// TIA Portal V17 export
// export: Created 2025-03-05T08:03:02.5022413Z, ExportSetting WithDefaults, DisplayName Totally Integrated Automation Portal, DisplayVersion V17 Update 8, DisplayName TIA Portal Openness, DisplayVersion V17 Update 8, DisplayName TIA Portal Version Control Interface, DisplayVersion V17, DisplayName SINAMICS Startdrive Advanced, DisplayVersion V17 SP2, DisplayName SINAMICS Startdrive G110M, G120, G120C, G120D, G120P, G115D, DisplayVersion V17 SP2, DisplayName SINAMICS Startdrive G130, G150, S120, S150, SINAMICS MV, S210, DisplayVersion V17 SP2, DisplayName STEP 7 Professional, DisplayVersion V17 Update 8, DisplayName SINUMERIK ONE STEP 7 Toolbox, DisplayVersion V17 Update 12, DisplayName SINUMERIK 840D sl STEP 7 Toolbox, DisplayVersion V17 Update 12, DisplayName STEP 7 Safety, DisplayVersion V17 Update 6, DisplayName WinCC Advanced, DisplayVersion V17 Update 8
FUNCTION "FC21012_POWDER_FEEDER_HEATER_JKL" : Void   // FC21012, LAD
TITLE = FC21012 POWDER FEEDER HEATER JKL
{ S7_Optimized_Access := 'TRUE' }
VERSION : 0.1
// stored: AutoNumber false, IsIECCheckEnabled false, SetENOAutomatically false, UDAEnableTagReadback false
BEGIN

REGION Network 1: /////_UNIT_01_/////
END_REGION

REGION Network 2: CALL FB21012 POWDER FEEDER 1 HEATER JKL UNIT 01
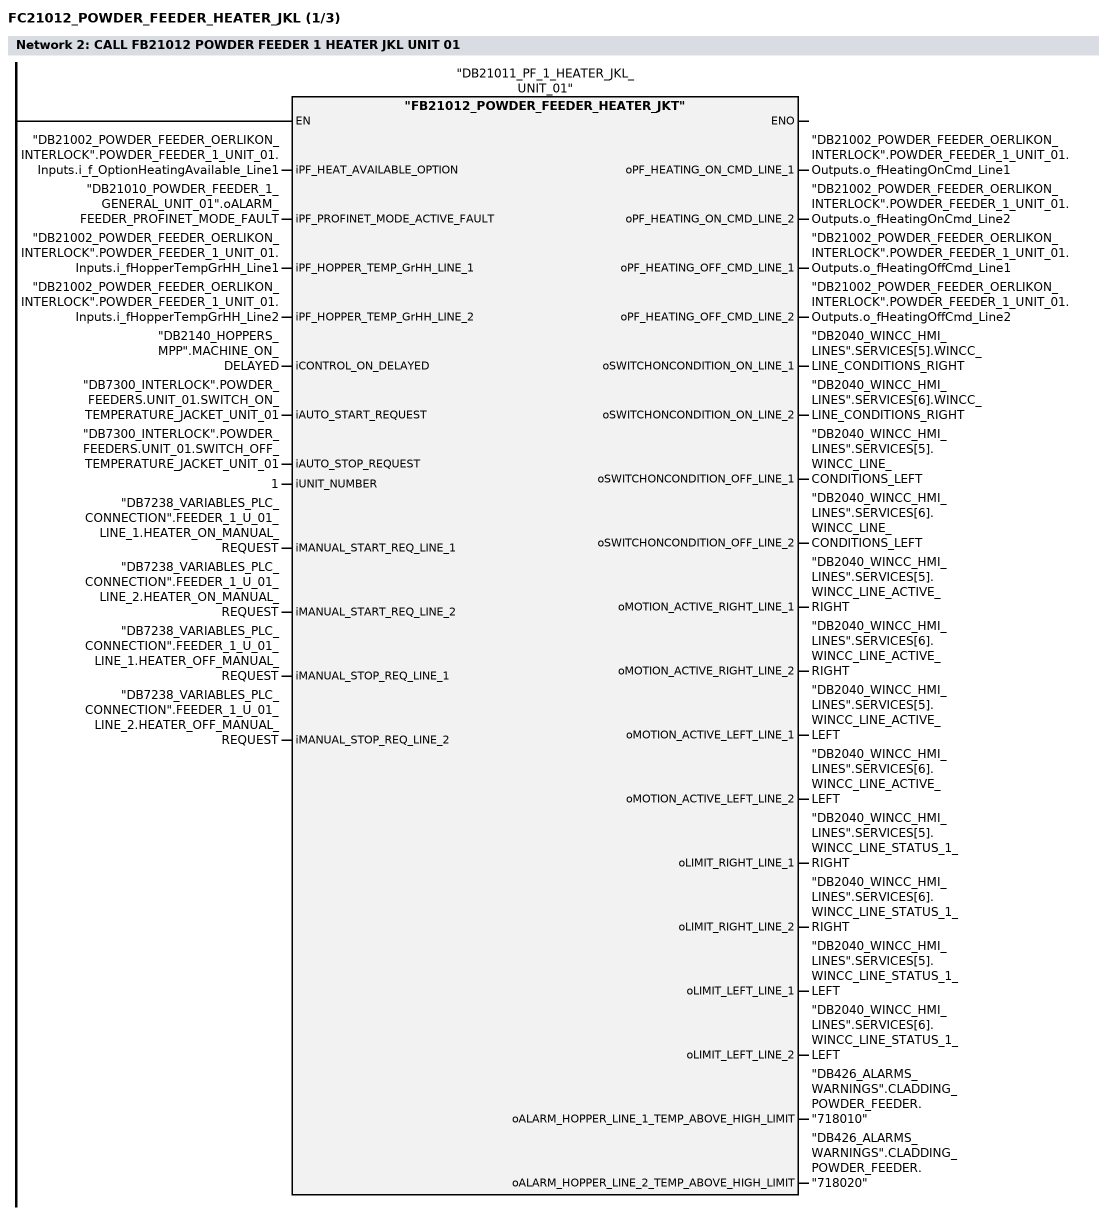
   RUNG wire#powerrail
      "DB21011_PF_1_HEATER_JKL_UNIT_01"(iPF_HEAT_AVAILABLE_OPTION := "DB21002_POWDER_FEEDER_OERLIKON_INTERLOCK".POWDER_FEEDER_1_UNIT_01.Inputs.i_f_OptionHeatingAvailable_Line1, iPF_PROFINET_MODE_ACTIVE_FAULT := "DB21010_POWDER_FEEDER_1_GENERAL_UNIT_01".oALARM_FEEDER_PROFINET_MODE_FAULT, iPF_HOPPER_TEMP_GrHH_LINE_1 := "DB21002_POWDER_FEEDER_OERLIKON_INTERLOCK".POWDER_FEEDER_1_UNIT_01.Inputs.i_fHopperTempGrHH_Line1, iPF_HOPPER_TEMP_GrHH_LINE_2 := "DB21002_POWDER_FEEDER_OERLIKON_INTERLOCK".POWDER_FEEDER_1_UNIT_01.Inputs.i_fHopperTempGrHH_Line2, iCONTROL_ON_DELAYED := "DB2140_HOPPERS_MPP".MACHINE_ON_DELAYED, iAUTO_START_REQUEST := "DB7300_INTERLOCK".POWDER_FEEDERS.UNIT_01.SWITCH_ON_TEMPERATURE_JACKET_UNIT_01, iAUTO_STOP_REQUEST := "DB7300_INTERLOCK".POWDER_FEEDERS.UNIT_01.SWITCH_OFF_TEMPERATURE_JACKET_UNIT_01, iUNIT_NUMBER := 1, iMANUAL_START_REQ_LINE_1 := "DB7238_VARIABLES_PLC_CONNECTION".FEEDER_1_U_01_LINE_1.HEATER_ON_MANUAL_REQUEST, iMANUAL_START_REQ_LINE_2 := "DB7238_VARIABLES_PLC_CONNECTION".FEEDER_1_U_01_LINE_2.HEATER_ON_MANUAL_REQUEST, iMANUAL_STOP_REQ_LINE_1 := "DB7238_VARIABLES_PLC_CONNECTION".FEEDER_1_U_01_LINE_1.HEATER_OFF_MANUAL_REQUEST, iMANUAL_STOP_REQ_LINE_2 := "DB7238_VARIABLES_PLC_CONNECTION".FEEDER_1_U_01_LINE_2.HEATER_OFF_MANUAL_REQUEST, oPF_HEATING_ON_CMD_LINE_1 => "DB21002_POWDER_FEEDER_OERLIKON_INTERLOCK".POWDER_FEEDER_1_UNIT_01.Outputs.o_fHeatingOnCmd_Line1, oPF_HEATING_ON_CMD_LINE_2 => "DB21002_POWDER_FEEDER_OERLIKON_INTERLOCK".POWDER_FEEDER_1_UNIT_01.Outputs.o_fHeatingOnCmd_Line2, oPF_HEATING_OFF_CMD_LINE_1 => "DB21002_POWDER_FEEDER_OERLIKON_INTERLOCK".POWDER_FEEDER_1_UNIT_01.Outputs.o_fHeatingOffCmd_Line1, oPF_HEATING_OFF_CMD_LINE_2 => "DB21002_POWDER_FEEDER_OERLIKON_INTERLOCK".POWDER_FEEDER_1_UNIT_01.Outputs.o_fHeatingOffCmd_Line2, oSWITCHONCONDITION_ON_LINE_1 => "DB2040_WINCC_HMI_LINES".SERVICES[5].WINCC_LINE_CONDITIONS_RIGHT, oSWITCHONCONDITION_ON_LINE_2 => "DB2040_WINCC_HMI_LINES".SERVICES[6].WINCC_LINE_CONDITIONS_RIGHT, oSWITCHONCONDITION_OFF_LINE_1 => "DB2040_WINCC_HMI_LINES".SERVICES[5].WINCC_LINE_CONDITIONS_LEFT, oSWITCHONCONDITION_OFF_LINE_2 => "DB2040_WINCC_HMI_LINES".SERVICES[6].WINCC_LINE_CONDITIONS_LEFT, oMOTION_ACTIVE_RIGHT_LINE_1 => "DB2040_WINCC_HMI_LINES".SERVICES[5].WINCC_LINE_ACTIVE_RIGHT, oMOTION_ACTIVE_RIGHT_LINE_2 => "DB2040_WINCC_HMI_LINES".SERVICES[6].WINCC_LINE_ACTIVE_RIGHT, oMOTION_ACTIVE_LEFT_LINE_1 => "DB2040_WINCC_HMI_LINES".SERVICES[5].WINCC_LINE_ACTIVE_LEFT, oMOTION_ACTIVE_LEFT_LINE_2 => "DB2040_WINCC_HMI_LINES".SERVICES[6].WINCC_LINE_ACTIVE_LEFT, oLIMIT_RIGHT_LINE_1 => "DB2040_WINCC_HMI_LINES".SERVICES[5].WINCC_LINE_STATUS_1_RIGHT, oLIMIT_RIGHT_LINE_2 => "DB2040_WINCC_HMI_LINES".SERVICES[6].WINCC_LINE_STATUS_1_RIGHT, oLIMIT_LEFT_LINE_1 => "DB2040_WINCC_HMI_LINES".SERVICES[5].WINCC_LINE_STATUS_1_LEFT, oLIMIT_LEFT_LINE_2 => "DB2040_WINCC_HMI_LINES".SERVICES[6].WINCC_LINE_STATUS_1_LEFT, oALARM_HOPPER_LINE_1_TEMP_ABOVE_HIGH_LIMIT => "DB426_ALARMS_WARNINGS".CLADDING_POWDER_FEEDER."718010", oALARM_HOPPER_LINE_2_TEMP_ABOVE_HIGH_LIMIT => "DB426_ALARMS_WARNINGS".CLADDING_POWDER_FEEDER."718020")
   END_RUNG
   // the same network as SCL:
   "DB21011_PF_1_HEATER_JKL_UNIT_01"(iPF_HEAT_AVAILABLE_OPTION := "DB21002_POWDER_FEEDER_OERLIKON_INTERLOCK".POWDER_FEEDER_1_UNIT_01.Inputs.i_f_OptionHeatingAvailable_Line1,   // "FB21012_POWDER_FEEDER_HEATER_JKT"
                           iPF_PROFINET_MODE_ACTIVE_FAULT := "DB21010_POWDER_FEEDER_1_GENERAL_UNIT_01".oALARM_FEEDER_PROFINET_MODE_FAULT,
                           iPF_HOPPER_TEMP_GrHH_LINE_1 := "DB21002_POWDER_FEEDER_OERLIKON_INTERLOCK".POWDER_FEEDER_1_UNIT_01.Inputs.i_fHopperTempGrHH_Line1,
                           iPF_HOPPER_TEMP_GrHH_LINE_2 := "DB21002_POWDER_FEEDER_OERLIKON_INTERLOCK".POWDER_FEEDER_1_UNIT_01.Inputs.i_fHopperTempGrHH_Line2,
                           iCONTROL_ON_DELAYED := "DB2140_HOPPERS_MPP".MACHINE_ON_DELAYED,
                           iAUTO_START_REQUEST := "DB7300_INTERLOCK".POWDER_FEEDERS.UNIT_01.SWITCH_ON_TEMPERATURE_JACKET_UNIT_01,
                           iAUTO_STOP_REQUEST := "DB7300_INTERLOCK".POWDER_FEEDERS.UNIT_01.SWITCH_OFF_TEMPERATURE_JACKET_UNIT_01,
                           iUNIT_NUMBER := 1,
                           iMANUAL_START_REQ_LINE_1 := "DB7238_VARIABLES_PLC_CONNECTION".FEEDER_1_U_01_LINE_1.HEATER_ON_MANUAL_REQUEST,
                           iMANUAL_START_REQ_LINE_2 := "DB7238_VARIABLES_PLC_CONNECTION".FEEDER_1_U_01_LINE_2.HEATER_ON_MANUAL_REQUEST,
                           iMANUAL_STOP_REQ_LINE_1 := "DB7238_VARIABLES_PLC_CONNECTION".FEEDER_1_U_01_LINE_1.HEATER_OFF_MANUAL_REQUEST,
                           iMANUAL_STOP_REQ_LINE_2 := "DB7238_VARIABLES_PLC_CONNECTION".FEEDER_1_U_01_LINE_2.HEATER_OFF_MANUAL_REQUEST,
                           oPF_HEATING_ON_CMD_LINE_1 => "DB21002_POWDER_FEEDER_OERLIKON_INTERLOCK".POWDER_FEEDER_1_UNIT_01.Outputs.o_fHeatingOnCmd_Line1,
                           oPF_HEATING_ON_CMD_LINE_2 => "DB21002_POWDER_FEEDER_OERLIKON_INTERLOCK".POWDER_FEEDER_1_UNIT_01.Outputs.o_fHeatingOnCmd_Line2,
                           oPF_HEATING_OFF_CMD_LINE_1 => "DB21002_POWDER_FEEDER_OERLIKON_INTERLOCK".POWDER_FEEDER_1_UNIT_01.Outputs.o_fHeatingOffCmd_Line1,
                           oPF_HEATING_OFF_CMD_LINE_2 => "DB21002_POWDER_FEEDER_OERLIKON_INTERLOCK".POWDER_FEEDER_1_UNIT_01.Outputs.o_fHeatingOffCmd_Line2,
                           oSWITCHONCONDITION_ON_LINE_1 => "DB2040_WINCC_HMI_LINES".SERVICES[5].WINCC_LINE_CONDITIONS_RIGHT,
                           oSWITCHONCONDITION_ON_LINE_2 => "DB2040_WINCC_HMI_LINES".SERVICES[6].WINCC_LINE_CONDITIONS_RIGHT,
                           oSWITCHONCONDITION_OFF_LINE_1 => "DB2040_WINCC_HMI_LINES".SERVICES[5].WINCC_LINE_CONDITIONS_LEFT,
                           oSWITCHONCONDITION_OFF_LINE_2 => "DB2040_WINCC_HMI_LINES".SERVICES[6].WINCC_LINE_CONDITIONS_LEFT,
                           oMOTION_ACTIVE_RIGHT_LINE_1 => "DB2040_WINCC_HMI_LINES".SERVICES[5].WINCC_LINE_ACTIVE_RIGHT,
                           oMOTION_ACTIVE_RIGHT_LINE_2 => "DB2040_WINCC_HMI_LINES".SERVICES[6].WINCC_LINE_ACTIVE_RIGHT,
                           oMOTION_ACTIVE_LEFT_LINE_1 => "DB2040_WINCC_HMI_LINES".SERVICES[5].WINCC_LINE_ACTIVE_LEFT,
                           oMOTION_ACTIVE_LEFT_LINE_2 => "DB2040_WINCC_HMI_LINES".SERVICES[6].WINCC_LINE_ACTIVE_LEFT,
                           oLIMIT_RIGHT_LINE_1 => "DB2040_WINCC_HMI_LINES".SERVICES[5].WINCC_LINE_STATUS_1_RIGHT,
                           oLIMIT_RIGHT_LINE_2 => "DB2040_WINCC_HMI_LINES".SERVICES[6].WINCC_LINE_STATUS_1_RIGHT,
                           oLIMIT_LEFT_LINE_1 => "DB2040_WINCC_HMI_LINES".SERVICES[5].WINCC_LINE_STATUS_1_LEFT,
                           oLIMIT_LEFT_LINE_2 => "DB2040_WINCC_HMI_LINES".SERVICES[6].WINCC_LINE_STATUS_1_LEFT,
                           oALARM_HOPPER_LINE_1_TEMP_ABOVE_HIGH_LIMIT => "DB426_ALARMS_WARNINGS".CLADDING_POWDER_FEEDER."718010",
                           oALARM_HOPPER_LINE_2_TEMP_ABOVE_HIGH_LIMIT => "DB426_ALARMS_WARNINGS".CLADDING_POWDER_FEEDER."718020");
END_REGION

REGION Network 3: /////_UNIT_02_/////
END_REGION

REGION Network 4: CALL FB21012 POWDER FEEDER 1 HEATER JKL UNIT 02
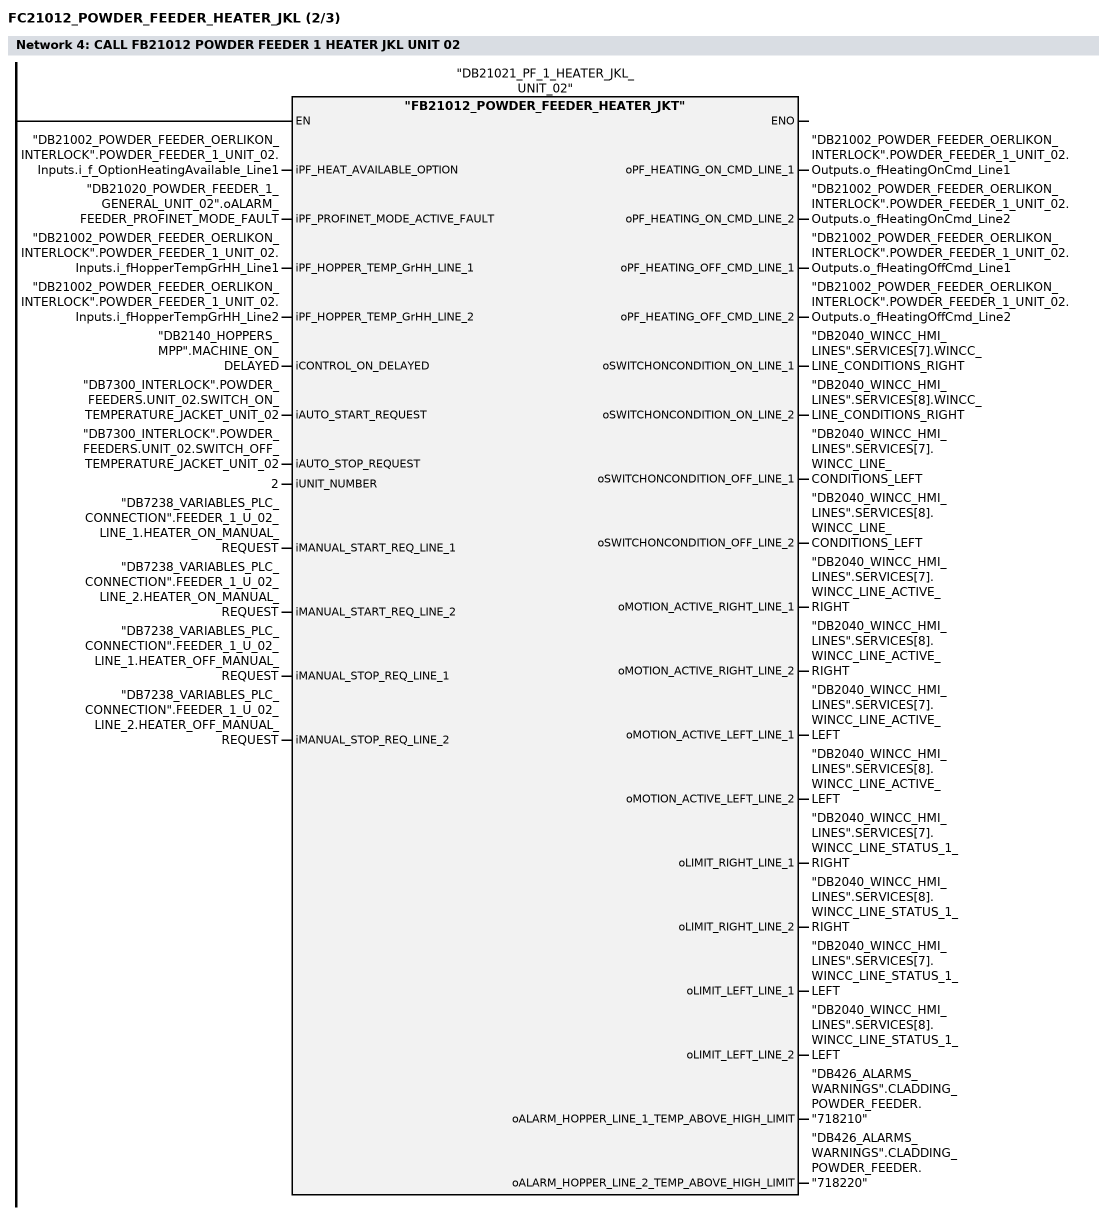
   RUNG wire#powerrail
      "DB21021_PF_1_HEATER_JKL_UNIT_02"(iPF_HEAT_AVAILABLE_OPTION := "DB21002_POWDER_FEEDER_OERLIKON_INTERLOCK".POWDER_FEEDER_1_UNIT_02.Inputs.i_f_OptionHeatingAvailable_Line1, iPF_PROFINET_MODE_ACTIVE_FAULT := "DB21020_POWDER_FEEDER_1_GENERAL_UNIT_02".oALARM_FEEDER_PROFINET_MODE_FAULT, iPF_HOPPER_TEMP_GrHH_LINE_1 := "DB21002_POWDER_FEEDER_OERLIKON_INTERLOCK".POWDER_FEEDER_1_UNIT_02.Inputs.i_fHopperTempGrHH_Line1, iPF_HOPPER_TEMP_GrHH_LINE_2 := "DB21002_POWDER_FEEDER_OERLIKON_INTERLOCK".POWDER_FEEDER_1_UNIT_02.Inputs.i_fHopperTempGrHH_Line2, iCONTROL_ON_DELAYED := "DB2140_HOPPERS_MPP".MACHINE_ON_DELAYED, iAUTO_START_REQUEST := "DB7300_INTERLOCK".POWDER_FEEDERS.UNIT_02.SWITCH_ON_TEMPERATURE_JACKET_UNIT_02, iAUTO_STOP_REQUEST := "DB7300_INTERLOCK".POWDER_FEEDERS.UNIT_02.SWITCH_OFF_TEMPERATURE_JACKET_UNIT_02, iUNIT_NUMBER := 2, iMANUAL_START_REQ_LINE_1 := "DB7238_VARIABLES_PLC_CONNECTION".FEEDER_1_U_02_LINE_1.HEATER_ON_MANUAL_REQUEST, iMANUAL_START_REQ_LINE_2 := "DB7238_VARIABLES_PLC_CONNECTION".FEEDER_1_U_02_LINE_2.HEATER_ON_MANUAL_REQUEST, iMANUAL_STOP_REQ_LINE_1 := "DB7238_VARIABLES_PLC_CONNECTION".FEEDER_1_U_02_LINE_1.HEATER_OFF_MANUAL_REQUEST, iMANUAL_STOP_REQ_LINE_2 := "DB7238_VARIABLES_PLC_CONNECTION".FEEDER_1_U_02_LINE_2.HEATER_OFF_MANUAL_REQUEST, oPF_HEATING_ON_CMD_LINE_1 => "DB21002_POWDER_FEEDER_OERLIKON_INTERLOCK".POWDER_FEEDER_1_UNIT_02.Outputs.o_fHeatingOnCmd_Line1, oPF_HEATING_ON_CMD_LINE_2 => "DB21002_POWDER_FEEDER_OERLIKON_INTERLOCK".POWDER_FEEDER_1_UNIT_02.Outputs.o_fHeatingOnCmd_Line2, oPF_HEATING_OFF_CMD_LINE_1 => "DB21002_POWDER_FEEDER_OERLIKON_INTERLOCK".POWDER_FEEDER_1_UNIT_02.Outputs.o_fHeatingOffCmd_Line1, oPF_HEATING_OFF_CMD_LINE_2 => "DB21002_POWDER_FEEDER_OERLIKON_INTERLOCK".POWDER_FEEDER_1_UNIT_02.Outputs.o_fHeatingOffCmd_Line2, oSWITCHONCONDITION_ON_LINE_1 => "DB2040_WINCC_HMI_LINES".SERVICES[7].WINCC_LINE_CONDITIONS_RIGHT, oSWITCHONCONDITION_ON_LINE_2 => "DB2040_WINCC_HMI_LINES".SERVICES[8].WINCC_LINE_CONDITIONS_RIGHT, oSWITCHONCONDITION_OFF_LINE_1 => "DB2040_WINCC_HMI_LINES".SERVICES[7].WINCC_LINE_CONDITIONS_LEFT, oSWITCHONCONDITION_OFF_LINE_2 => "DB2040_WINCC_HMI_LINES".SERVICES[8].WINCC_LINE_CONDITIONS_LEFT, oMOTION_ACTIVE_RIGHT_LINE_1 => "DB2040_WINCC_HMI_LINES".SERVICES[7].WINCC_LINE_ACTIVE_RIGHT, oMOTION_ACTIVE_RIGHT_LINE_2 => "DB2040_WINCC_HMI_LINES".SERVICES[8].WINCC_LINE_ACTIVE_RIGHT, oMOTION_ACTIVE_LEFT_LINE_1 => "DB2040_WINCC_HMI_LINES".SERVICES[7].WINCC_LINE_ACTIVE_LEFT, oMOTION_ACTIVE_LEFT_LINE_2 => "DB2040_WINCC_HMI_LINES".SERVICES[8].WINCC_LINE_ACTIVE_LEFT, oLIMIT_RIGHT_LINE_1 => "DB2040_WINCC_HMI_LINES".SERVICES[7].WINCC_LINE_STATUS_1_RIGHT, oLIMIT_RIGHT_LINE_2 => "DB2040_WINCC_HMI_LINES".SERVICES[8].WINCC_LINE_STATUS_1_RIGHT, oLIMIT_LEFT_LINE_1 => "DB2040_WINCC_HMI_LINES".SERVICES[7].WINCC_LINE_STATUS_1_LEFT, oLIMIT_LEFT_LINE_2 => "DB2040_WINCC_HMI_LINES".SERVICES[8].WINCC_LINE_STATUS_1_LEFT, oALARM_HOPPER_LINE_1_TEMP_ABOVE_HIGH_LIMIT => "DB426_ALARMS_WARNINGS".CLADDING_POWDER_FEEDER."718210", oALARM_HOPPER_LINE_2_TEMP_ABOVE_HIGH_LIMIT => "DB426_ALARMS_WARNINGS".CLADDING_POWDER_FEEDER."718220")
   END_RUNG
   // the same network as SCL:
   "DB21021_PF_1_HEATER_JKL_UNIT_02"(iPF_HEAT_AVAILABLE_OPTION := "DB21002_POWDER_FEEDER_OERLIKON_INTERLOCK".POWDER_FEEDER_1_UNIT_02.Inputs.i_f_OptionHeatingAvailable_Line1,   // "FB21012_POWDER_FEEDER_HEATER_JKT"
                           iPF_PROFINET_MODE_ACTIVE_FAULT := "DB21020_POWDER_FEEDER_1_GENERAL_UNIT_02".oALARM_FEEDER_PROFINET_MODE_FAULT,
                           iPF_HOPPER_TEMP_GrHH_LINE_1 := "DB21002_POWDER_FEEDER_OERLIKON_INTERLOCK".POWDER_FEEDER_1_UNIT_02.Inputs.i_fHopperTempGrHH_Line1,
                           iPF_HOPPER_TEMP_GrHH_LINE_2 := "DB21002_POWDER_FEEDER_OERLIKON_INTERLOCK".POWDER_FEEDER_1_UNIT_02.Inputs.i_fHopperTempGrHH_Line2,
                           iCONTROL_ON_DELAYED := "DB2140_HOPPERS_MPP".MACHINE_ON_DELAYED,
                           iAUTO_START_REQUEST := "DB7300_INTERLOCK".POWDER_FEEDERS.UNIT_02.SWITCH_ON_TEMPERATURE_JACKET_UNIT_02,
                           iAUTO_STOP_REQUEST := "DB7300_INTERLOCK".POWDER_FEEDERS.UNIT_02.SWITCH_OFF_TEMPERATURE_JACKET_UNIT_02,
                           iUNIT_NUMBER := 2,
                           iMANUAL_START_REQ_LINE_1 := "DB7238_VARIABLES_PLC_CONNECTION".FEEDER_1_U_02_LINE_1.HEATER_ON_MANUAL_REQUEST,
                           iMANUAL_START_REQ_LINE_2 := "DB7238_VARIABLES_PLC_CONNECTION".FEEDER_1_U_02_LINE_2.HEATER_ON_MANUAL_REQUEST,
                           iMANUAL_STOP_REQ_LINE_1 := "DB7238_VARIABLES_PLC_CONNECTION".FEEDER_1_U_02_LINE_1.HEATER_OFF_MANUAL_REQUEST,
                           iMANUAL_STOP_REQ_LINE_2 := "DB7238_VARIABLES_PLC_CONNECTION".FEEDER_1_U_02_LINE_2.HEATER_OFF_MANUAL_REQUEST,
                           oPF_HEATING_ON_CMD_LINE_1 => "DB21002_POWDER_FEEDER_OERLIKON_INTERLOCK".POWDER_FEEDER_1_UNIT_02.Outputs.o_fHeatingOnCmd_Line1,
                           oPF_HEATING_ON_CMD_LINE_2 => "DB21002_POWDER_FEEDER_OERLIKON_INTERLOCK".POWDER_FEEDER_1_UNIT_02.Outputs.o_fHeatingOnCmd_Line2,
                           oPF_HEATING_OFF_CMD_LINE_1 => "DB21002_POWDER_FEEDER_OERLIKON_INTERLOCK".POWDER_FEEDER_1_UNIT_02.Outputs.o_fHeatingOffCmd_Line1,
                           oPF_HEATING_OFF_CMD_LINE_2 => "DB21002_POWDER_FEEDER_OERLIKON_INTERLOCK".POWDER_FEEDER_1_UNIT_02.Outputs.o_fHeatingOffCmd_Line2,
                           oSWITCHONCONDITION_ON_LINE_1 => "DB2040_WINCC_HMI_LINES".SERVICES[7].WINCC_LINE_CONDITIONS_RIGHT,
                           oSWITCHONCONDITION_ON_LINE_2 => "DB2040_WINCC_HMI_LINES".SERVICES[8].WINCC_LINE_CONDITIONS_RIGHT,
                           oSWITCHONCONDITION_OFF_LINE_1 => "DB2040_WINCC_HMI_LINES".SERVICES[7].WINCC_LINE_CONDITIONS_LEFT,
                           oSWITCHONCONDITION_OFF_LINE_2 => "DB2040_WINCC_HMI_LINES".SERVICES[8].WINCC_LINE_CONDITIONS_LEFT,
                           oMOTION_ACTIVE_RIGHT_LINE_1 => "DB2040_WINCC_HMI_LINES".SERVICES[7].WINCC_LINE_ACTIVE_RIGHT,
                           oMOTION_ACTIVE_RIGHT_LINE_2 => "DB2040_WINCC_HMI_LINES".SERVICES[8].WINCC_LINE_ACTIVE_RIGHT,
                           oMOTION_ACTIVE_LEFT_LINE_1 => "DB2040_WINCC_HMI_LINES".SERVICES[7].WINCC_LINE_ACTIVE_LEFT,
                           oMOTION_ACTIVE_LEFT_LINE_2 => "DB2040_WINCC_HMI_LINES".SERVICES[8].WINCC_LINE_ACTIVE_LEFT,
                           oLIMIT_RIGHT_LINE_1 => "DB2040_WINCC_HMI_LINES".SERVICES[7].WINCC_LINE_STATUS_1_RIGHT,
                           oLIMIT_RIGHT_LINE_2 => "DB2040_WINCC_HMI_LINES".SERVICES[8].WINCC_LINE_STATUS_1_RIGHT,
                           oLIMIT_LEFT_LINE_1 => "DB2040_WINCC_HMI_LINES".SERVICES[7].WINCC_LINE_STATUS_1_LEFT,
                           oLIMIT_LEFT_LINE_2 => "DB2040_WINCC_HMI_LINES".SERVICES[8].WINCC_LINE_STATUS_1_LEFT,
                           oALARM_HOPPER_LINE_1_TEMP_ABOVE_HIGH_LIMIT => "DB426_ALARMS_WARNINGS".CLADDING_POWDER_FEEDER."718210",
                           oALARM_HOPPER_LINE_2_TEMP_ABOVE_HIGH_LIMIT => "DB426_ALARMS_WARNINGS".CLADDING_POWDER_FEEDER."718220");
END_REGION

REGION Network 5: CALL FB21012 POWDER FEEDER 2 HEATER JKL UNIT 02
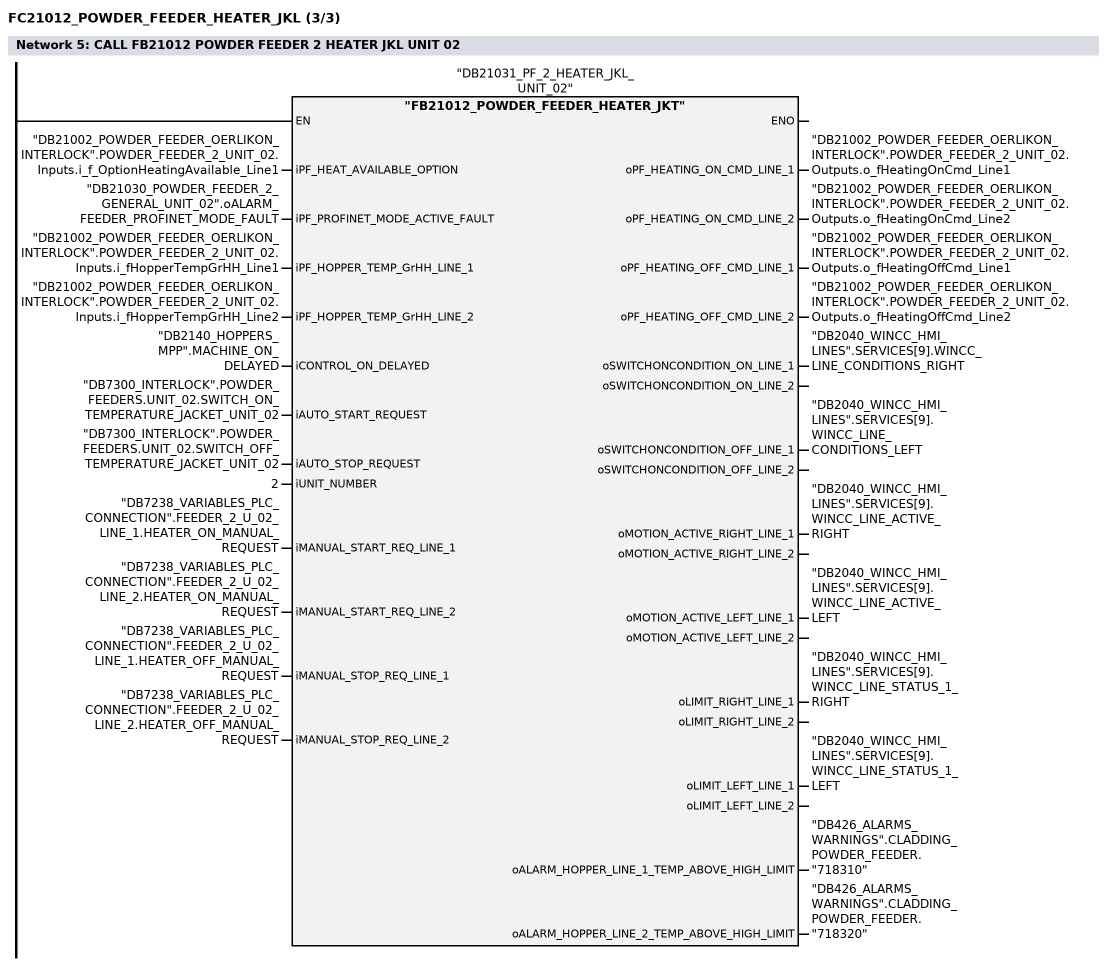
   RUNG wire#powerrail
      "DB21031_PF_2_HEATER_JKL_UNIT_02"(iPF_HEAT_AVAILABLE_OPTION := "DB21002_POWDER_FEEDER_OERLIKON_INTERLOCK".POWDER_FEEDER_2_UNIT_02.Inputs.i_f_OptionHeatingAvailable_Line1, iPF_PROFINET_MODE_ACTIVE_FAULT := "DB21030_POWDER_FEEDER_2_GENERAL_UNIT_02".oALARM_FEEDER_PROFINET_MODE_FAULT, iPF_HOPPER_TEMP_GrHH_LINE_1 := "DB21002_POWDER_FEEDER_OERLIKON_INTERLOCK".POWDER_FEEDER_2_UNIT_02.Inputs.i_fHopperTempGrHH_Line1, iPF_HOPPER_TEMP_GrHH_LINE_2 := "DB21002_POWDER_FEEDER_OERLIKON_INTERLOCK".POWDER_FEEDER_2_UNIT_02.Inputs.i_fHopperTempGrHH_Line2, iCONTROL_ON_DELAYED := "DB2140_HOPPERS_MPP".MACHINE_ON_DELAYED, iAUTO_START_REQUEST := "DB7300_INTERLOCK".POWDER_FEEDERS.UNIT_02.SWITCH_ON_TEMPERATURE_JACKET_UNIT_02, iAUTO_STOP_REQUEST := "DB7300_INTERLOCK".POWDER_FEEDERS.UNIT_02.SWITCH_OFF_TEMPERATURE_JACKET_UNIT_02, iUNIT_NUMBER := 2, iMANUAL_START_REQ_LINE_1 := "DB7238_VARIABLES_PLC_CONNECTION".FEEDER_2_U_02_LINE_1.HEATER_ON_MANUAL_REQUEST, iMANUAL_START_REQ_LINE_2 := "DB7238_VARIABLES_PLC_CONNECTION".FEEDER_2_U_02_LINE_2.HEATER_ON_MANUAL_REQUEST, iMANUAL_STOP_REQ_LINE_1 := "DB7238_VARIABLES_PLC_CONNECTION".FEEDER_2_U_02_LINE_1.HEATER_OFF_MANUAL_REQUEST, iMANUAL_STOP_REQ_LINE_2 := "DB7238_VARIABLES_PLC_CONNECTION".FEEDER_2_U_02_LINE_2.HEATER_OFF_MANUAL_REQUEST, oPF_HEATING_ON_CMD_LINE_1 => "DB21002_POWDER_FEEDER_OERLIKON_INTERLOCK".POWDER_FEEDER_2_UNIT_02.Outputs.o_fHeatingOnCmd_Line1, oPF_HEATING_ON_CMD_LINE_2 => "DB21002_POWDER_FEEDER_OERLIKON_INTERLOCK".POWDER_FEEDER_2_UNIT_02.Outputs.o_fHeatingOnCmd_Line2, oPF_HEATING_OFF_CMD_LINE_1 => "DB21002_POWDER_FEEDER_OERLIKON_INTERLOCK".POWDER_FEEDER_2_UNIT_02.Outputs.o_fHeatingOffCmd_Line1, oPF_HEATING_OFF_CMD_LINE_2 => "DB21002_POWDER_FEEDER_OERLIKON_INTERLOCK".POWDER_FEEDER_2_UNIT_02.Outputs.o_fHeatingOffCmd_Line2, oSWITCHONCONDITION_ON_LINE_1 => "DB2040_WINCC_HMI_LINES".SERVICES[9].WINCC_LINE_CONDITIONS_RIGHT, oSWITCHONCONDITION_ON_LINE_2 =>, oSWITCHONCONDITION_OFF_LINE_1 => "DB2040_WINCC_HMI_LINES".SERVICES[9].WINCC_LINE_CONDITIONS_LEFT, oSWITCHONCONDITION_OFF_LINE_2 =>, oMOTION_ACTIVE_RIGHT_LINE_1 => "DB2040_WINCC_HMI_LINES".SERVICES[9].WINCC_LINE_ACTIVE_RIGHT, oMOTION_ACTIVE_RIGHT_LINE_2 =>, oMOTION_ACTIVE_LEFT_LINE_1 => "DB2040_WINCC_HMI_LINES".SERVICES[9].WINCC_LINE_ACTIVE_LEFT, oMOTION_ACTIVE_LEFT_LINE_2 =>, oLIMIT_RIGHT_LINE_1 => "DB2040_WINCC_HMI_LINES".SERVICES[9].WINCC_LINE_STATUS_1_RIGHT, oLIMIT_RIGHT_LINE_2 =>, oLIMIT_LEFT_LINE_1 => "DB2040_WINCC_HMI_LINES".SERVICES[9].WINCC_LINE_STATUS_1_LEFT, oLIMIT_LEFT_LINE_2 =>, oALARM_HOPPER_LINE_1_TEMP_ABOVE_HIGH_LIMIT => "DB426_ALARMS_WARNINGS".CLADDING_POWDER_FEEDER."718310", oALARM_HOPPER_LINE_2_TEMP_ABOVE_HIGH_LIMIT => "DB426_ALARMS_WARNINGS".CLADDING_POWDER_FEEDER."718320")
   END_RUNG
   // the same network as SCL:
   "DB21031_PF_2_HEATER_JKL_UNIT_02"(iPF_HEAT_AVAILABLE_OPTION := "DB21002_POWDER_FEEDER_OERLIKON_INTERLOCK".POWDER_FEEDER_2_UNIT_02.Inputs.i_f_OptionHeatingAvailable_Line1,   // "FB21012_POWDER_FEEDER_HEATER_JKT"
                           iPF_PROFINET_MODE_ACTIVE_FAULT := "DB21030_POWDER_FEEDER_2_GENERAL_UNIT_02".oALARM_FEEDER_PROFINET_MODE_FAULT,
                           iPF_HOPPER_TEMP_GrHH_LINE_1 := "DB21002_POWDER_FEEDER_OERLIKON_INTERLOCK".POWDER_FEEDER_2_UNIT_02.Inputs.i_fHopperTempGrHH_Line1,
                           iPF_HOPPER_TEMP_GrHH_LINE_2 := "DB21002_POWDER_FEEDER_OERLIKON_INTERLOCK".POWDER_FEEDER_2_UNIT_02.Inputs.i_fHopperTempGrHH_Line2,
                           iCONTROL_ON_DELAYED := "DB2140_HOPPERS_MPP".MACHINE_ON_DELAYED,
                           iAUTO_START_REQUEST := "DB7300_INTERLOCK".POWDER_FEEDERS.UNIT_02.SWITCH_ON_TEMPERATURE_JACKET_UNIT_02,
                           iAUTO_STOP_REQUEST := "DB7300_INTERLOCK".POWDER_FEEDERS.UNIT_02.SWITCH_OFF_TEMPERATURE_JACKET_UNIT_02,
                           iUNIT_NUMBER := 2,
                           iMANUAL_START_REQ_LINE_1 := "DB7238_VARIABLES_PLC_CONNECTION".FEEDER_2_U_02_LINE_1.HEATER_ON_MANUAL_REQUEST,
                           iMANUAL_START_REQ_LINE_2 := "DB7238_VARIABLES_PLC_CONNECTION".FEEDER_2_U_02_LINE_2.HEATER_ON_MANUAL_REQUEST,
                           iMANUAL_STOP_REQ_LINE_1 := "DB7238_VARIABLES_PLC_CONNECTION".FEEDER_2_U_02_LINE_1.HEATER_OFF_MANUAL_REQUEST,
                           iMANUAL_STOP_REQ_LINE_2 := "DB7238_VARIABLES_PLC_CONNECTION".FEEDER_2_U_02_LINE_2.HEATER_OFF_MANUAL_REQUEST,
                           oPF_HEATING_ON_CMD_LINE_1 => "DB21002_POWDER_FEEDER_OERLIKON_INTERLOCK".POWDER_FEEDER_2_UNIT_02.Outputs.o_fHeatingOnCmd_Line1,
                           oPF_HEATING_ON_CMD_LINE_2 => "DB21002_POWDER_FEEDER_OERLIKON_INTERLOCK".POWDER_FEEDER_2_UNIT_02.Outputs.o_fHeatingOnCmd_Line2,
                           oPF_HEATING_OFF_CMD_LINE_1 => "DB21002_POWDER_FEEDER_OERLIKON_INTERLOCK".POWDER_FEEDER_2_UNIT_02.Outputs.o_fHeatingOffCmd_Line1,
                           oPF_HEATING_OFF_CMD_LINE_2 => "DB21002_POWDER_FEEDER_OERLIKON_INTERLOCK".POWDER_FEEDER_2_UNIT_02.Outputs.o_fHeatingOffCmd_Line2,
                           oSWITCHONCONDITION_ON_LINE_1 => "DB2040_WINCC_HMI_LINES".SERVICES[9].WINCC_LINE_CONDITIONS_RIGHT,
                           oSWITCHONCONDITION_OFF_LINE_1 => "DB2040_WINCC_HMI_LINES".SERVICES[9].WINCC_LINE_CONDITIONS_LEFT,
                           oMOTION_ACTIVE_RIGHT_LINE_1 => "DB2040_WINCC_HMI_LINES".SERVICES[9].WINCC_LINE_ACTIVE_RIGHT,
                           oMOTION_ACTIVE_LEFT_LINE_1 => "DB2040_WINCC_HMI_LINES".SERVICES[9].WINCC_LINE_ACTIVE_LEFT,
                           oLIMIT_RIGHT_LINE_1 => "DB2040_WINCC_HMI_LINES".SERVICES[9].WINCC_LINE_STATUS_1_RIGHT,
                           oLIMIT_LEFT_LINE_1 => "DB2040_WINCC_HMI_LINES".SERVICES[9].WINCC_LINE_STATUS_1_LEFT,
                           oALARM_HOPPER_LINE_1_TEMP_ABOVE_HIGH_LIMIT => "DB426_ALARMS_WARNINGS".CLADDING_POWDER_FEEDER."718310",
                           oALARM_HOPPER_LINE_2_TEMP_ABOVE_HIGH_LIMIT => "DB426_ALARMS_WARNINGS".CLADDING_POWDER_FEEDER."718320");
END_REGION
END_FUNCTION
